INTERFACE Collection

METHOD createIterator : Iterator
VAR_INPUT
END_VAR
END_METHOD

END_INTERFACE

(* stored: Version 1.1.0.1, ProductVersion 3.1.4024.12
   Itf Collection: Id {6730e63c-3da3-432d-8c54-aa42ffee9239}
   Method createIterator: Id {89d6281e-62b2-4f2a-8e6f-4afeed93e2c0} *)
